TYPE E_GaugeState :
(
	Valid := gc_GaugeValidState,
	ValidHi	:= 1, //gc_GaugeValidState + 1,
	ValidLo	:= 2, //gc_GaugeValidState + 2,
	
	// Invalid states
	Invalid	:= -1, //gc_GaugeValidState - 1,
	Disconnected	:=	-2, //gc_GaugeValidState -2,
	OoR	:= -6, //gc_GaugeValidState -6,
	// Ion gauges
	Off		:= -3, //gc_GaugeValidState - 3,
	Starting	:= -4 //gc_GaugeValidState - 4
) INT;
END_TYPE

(* stored: Version 1.1.0.1, ProductVersion 3.1.4018.5
   DUT E_GaugeState: Id {c25a9601-e125-4f1e-8734-ed2a641d27b1} *)
